KUKA KRL data list: tcp_chk_1.dat

&ACCESS RVP
&REL 151
&COMMENT TCP CHECK TOOL 1
DEFDAT  TCP_CHK_1
;FOLD EXTERNAL DECLARATIONS;%{PE}%V3.2.0,%MKUKATPBASIS,%CEXT,%VCOMMON,%P
;FOLD GRIPPERTECH EXT
EXT  H50 (INT  :IN,INT  :IN,INT  :IN,GRP_TYP  :IN )
;ENDFOLD (GRIPPERTECH EXT)
;FOLD SPOTTECH EXT
EXT  USERSPOT (S_COMMAND  :IN,SPOT_TYPE  :IN )
;ENDFOLD (SPOTTECH EXT)
;FOLD BAS EXT;%{PE}%V3.2.0,%MKUKATPBASIS,%CEXT,%VEXT,%P
EXT  BAS (BAS_COMMAND  :IN,REAL  :IN )
DECL INT SUCCESS
;ENDFOLD
;FOLD USER EXT;%{E}%V3.2.0,%MKUKATPUSER,%CEXT,%VEXT,%P
;Make here your modifications
;ENDFOLD
;ENDFOLD
;FOLD USER EXT;%{}%V2.2.2,%MKUKATPUSER,%CEXT,%VEXT,%P
;Make here your modifications
DECL BOOL TIPKONTROLE
DECL INT ANSWER
DECL INT WAITTIME=1000
;ENDFOLD
;ENDFOLD
DECL INT I
;*      FDAT Declarations     *

;******************************
;*     E6POS Declarations     *
;******************************

DECL E6POS XP10={X 1991.58301,Y -779.688782,Z 1569.90405,A -142.057907,B 56.2479897,C -135.499695,S 2,T 2,E1 0.0,E2 0.0,E3 0.0,E4 0.0,E5 0.0,E6 0.0}
DECL E6POS XSERV_POS_1={X 84.4434509,Y 1847.146,Z 1622.83398,A 86.5612411,B -12.4712801,C -179.259094,S 6,T 27,E1 -1563.58301,E2 0.0,E3 0.0,E4 0.0,E5 0.0,E6 0.0}
DECL E6POS XP20={X 1368.17004,Y -1604.78003,Z 695.290527,A -176.796097,B 21.8214397,C -158.206604,S 2,T 2,E1 0.0,E2 0.0,E3 0.0,E4 0.0,E5 0.0,E6 0.0}

;******************************
;*     FDAT Declarations      *
;******************************

DECL FDAT FP10={TOOL_NO 14,BASE_NO 0,IPO_FRAME #BASE,TQ_STATE FALSE}
DECL FDAT FSERV_POS_1={TOOL_NO 1,BASE_NO 0,IPO_FRAME #BASE}
DECL FDAT FP20={TOOL_NO 14,BASE_NO 0,IPO_FRAME #BASE,TQ_STATE FALSE}

;******************************
;*  PDAT & LDAT Declarations  *
;******************************

DECL PDAT PH={VEL 100.0,ACC 100.0,APO_DIST 100.0,APO_MODE #CPTP}

DECL E6POS XP30={X 2311.08911,Y -615.218384,Z 582.254517,A 52.0533791,B 11.4944496,C -0.662933111,S 2,T 10,E1 -367.19989,E2 0.0,E3 0.0,E4 0.0,E5 0.0,E6 0.0}
DECL FDAT FP30={TOOL_NO 1,BASE_NO 0,IPO_FRAME #BASE,POINT2[] " "}
DECL E6POS XP40={X 2415.06006,Y -661.647217,Z -64.6423798,A 52.025631,B 13.8356104,C -0.669203103,S 2,T 8,E1 -367.19989,E2 0.0,E3 0.0,E4 0.0,E5 0.0,E6 0.0}
DECL FDAT FP40={TOOL_NO 1,BASE_NO 0,IPO_FRAME #BASE,POINT2[] " "}
DECL E6POS XP50={X 1079.88,Y -976.492493,Z 903.200806,A -177.984299,B 18.5442696,C -161.646393,S 2,T 2,E1 0.0,E2 0.0,E3 0.0,E4 0.0,E5 0.0,E6 0.0}
DECL FDAT FP50={TOOL_NO 0,BASE_NO 0,IPO_FRAME #BASE,POINT2[] " ",TQ_STATE FALSE}
DECL E6POS XP60={X 1368.17004,Y -1604.78003,Z 695.290527,A -176.796097,B 21.8214397,C -158.206604,S 2,T 2,E1 0.0,E2 0.0,E3 0.0,E4 0.0,E5 0.0,E6 0.0}
DECL FDAT FP60={TOOL_NO 14,BASE_NO 0,IPO_FRAME #BASE,POINT2[] " ",TQ_STATE FALSE}
DECL E6POS XP70={X 1991.58301,Y -779.688782,Z 1569.90405,A -142.057907,B 56.2479897,C -135.499695,S 2,T 2,E1 0.0,E2 0.0,E3 0.0,E4 0.0,E5 0.0,E6 0.0}
DECL FDAT FP70={TOOL_NO 14,BASE_NO 0,IPO_FRAME #BASE,POINT2[] " ",TQ_STATE FALSE}
DECL E6POS XP80={X 2192.04395,Y -596.577576,Z 555.076416,A -14.5445995,B 80.1722412,C -56.6474991,S 2,T 10,E1 -367.19989,E2 0.0,E3 0.0,E4 0.0,E5 0.0,E6 0.0}
DECL FDAT FP80={TOOL_NO 1,BASE_NO 0,IPO_FRAME #BASE,POINT2[] " "}
DECL E6POS XTCP_CHK_POSITION={X 84.4434509,Y 1847.146,Z 1622.83398,A 86.5612411,B -12.4712801,C -179.259094,S 6,T 27,E1 -1563.58301,E2 0.0,E3 0.0,E4 0.0,E5 0.0,E6 0.0}
DECL FDAT FTCP_CHK_POSITION={TOOL_NO 1,BASE_NO 0,IPO_FRAME #BASE,POINT2[] " "}
DECL E6POS XTCP_CHK_POS_1={X 818.403015,Y -1651.55701,Z -109.656601,A 172.554398,B -1.01382303,C -179.870605,S 2,T 2,E1 0.0,E2 0.0,E3 0.0,E4 0.0,E5 0.0,E6 0.0}
DECL FDAT FTCP_CHK_POS_1={TOOL_NO 14,BASE_NO 0,IPO_FRAME #BASE,POINT2[] " ",TQ_STATE FALSE}
DECL E6POS XP41={X 2432.96289,Y -476.577606,Z -71.2344208,A 52.0531807,B 11.4962101,C -0.664697111,S 2,T 8,E1 -367.19989,E2 0.0,E3 0.0,E4 0.0,E5 0.0,E6 0.0}
DECL FDAT FP41={TOOL_NO 1,BASE_NO 0,IPO_FRAME #BASE,POINT2[] " "}
DECL E6POS XP81={X 1822.90698,Y -654.884888,Z 640.681885,A 41.8054695,B 56.6090698,C 47.6876106,S 6,T 26,E1 -1972.61694,E2 0.0,E3 0.0,E4 0.0,E5 0.0,E6 0.0}
DECL FDAT FP81={TOOL_NO 1,BASE_NO 0,IPO_FRAME #BASE,POINT2[] " "}
DECL E6POS XBefore_Check_Point_1={X 818.62738,Y -1651.66101,Z -32.1126099,A 172.352905,B -1.31993604,C -179.733002,S 2,T 2,E1 0.0,E2 0.0,E3 0.0,E4 0.0,E5 0.0,E6 0.0}
DECL FDAT FBefore_Check_Point_1={TOOL_NO 14,BASE_NO 0,IPO_FRAME #BASE,POINT2[] " ",TQ_STATE FALSE}
DECL LDAT LH={VEL 2.0,ACC 100.0,APO_DIST 100.0,APO_FAC 50.0,ORI_TYP #VAR}
DECL E6POS XAFTER_CHECK_POINT_1={X 818.401428,Y -1651.55701,Z 10.4140701,A 172.554199,B -1.01384497,C -179.870697,S 2,T 2,E1 0.0,E2 0.0,E3 0.0,E4 0.0,E5 0.0,E6 0.0}
DECL FDAT FAfter_Check_Point_1={TOOL_NO 14,BASE_NO 0,IPO_FRAME #BASE,POINT2[] " ",TQ_STATE FALSE}
DECL E6POS XP75={X 2305.34692,Y -723.78302,Z 579.621582,A -14.5605898,B 80.1713333,C -56.66325,S 2,T 10,E1 -367.19989,E2 0.0,E3 0.0,E4 0.0,E5 0.0,E6 0.0}
DECL FDAT FP75={TOOL_NO 1,BASE_NO 0,IPO_FRAME #BASE,POINT2[] " "}
DECL E6POS XP90={X 2410.20093,Y -416.701294,Z 388.115906,A -122.975998,B 80.2214584,C -160.4422,S 2,T 10,E1 -422.983612,E2 0.0,E3 0.0,E4 0.0,E5 0.0,E6 0.0}
DECL FDAT FP90={TOOL_NO 1,BASE_NO 0,IPO_FRAME #BASE,POINT2[] " "}
DECL E6POS XBefore_Check_Point_2={X 2377.53491,Y -467.046295,Z 39.8671989,A -122.976303,B 80.2215729,C -160.442596,S 2,T 10,E1 -422.983612,E2 0.0,E3 0.0,E4 0.0,E5 0.0,E6 0.0}
DECL FDAT FBefore_Check_Point_2={TOOL_NO 1,BASE_NO 0,IPO_FRAME #BASE,POINT2[] " "}
DECL E6POS XTCP_CHK_POS_2={X 2426.96411,Y -429.442688,Z 29.7570896,A -126.074799,B 78.3430786,C -164.518799,S 2,T 10,E1 -422.981812,E2 0.0,E3 0.0,E4 0.0,E5 0.0,E6 0.0}
DECL FDAT FTCP_CHK_POS_2={TOOL_NO 1,BASE_NO 0,IPO_FRAME #BASE,POINT2[] " "}
DECL E6POS XAfter_Check_Point_2={X 2377.53491,Y -467.046295,Z 39.8671989,A -122.976303,B 80.2215729,C -160.442596,S 2,T 10,E1 -422.983612,E2 0.0,E3 0.0,E4 0.0,E5 0.0,E6 0.0}
DECL FDAT FAfter_Check_Point_2={TOOL_NO 1,BASE_NO 0,IPO_FRAME #BASE,POINT2[] " "}
DECL E6POS XP100={X 2410.19995,Y -416.696594,Z 388.11441,A -122.976501,B 80.2214966,C -160.442795,S 2,T 10,E1 -422.985291,E2 0.0,E3 0.0,E4 0.0,E5 0.0,E6 0.0}
DECL FDAT FP100={TOOL_NO 1,BASE_NO 0,IPO_FRAME #BASE,POINT2[] " "}
DECL E6POS XP110={X 1784.026,Y -939.821716,Z 564.808594,A -112.103302,B 88.3751907,C -136.251404,S 2,T 10,E1 -586.802917,E2 0.0,E3 0.0,E4 0.0,E5 0.0,E6 0.0}
DECL FDAT FP110={TOOL_NO 1,BASE_NO 0,IPO_FRAME #BASE,POINT2[] " "}
DECL E6POS XP120={X 996.789307,Y -1256.22302,Z 985.020386,A -19.8349094,B 83.8573227,C -28.9672508,S 2,T 10,E1 -831.47522,E2 0.0,E3 0.0,E4 0.0,E5 0.0,E6 0.0}
DECL FDAT FP120={TOOL_NO 1,BASE_NO 0,IPO_FRAME #BASE,POINT2[] " "}
DECL E6POS XP130={X 605.816284,Y -317.149902,Z 1161.85999,A 86.4495468,B 72.0065536,C 88.4566193,S 6,T 26,E1 -1309.93506,E2 0.0,E3 0.0,E4 0.0,E5 0.0,E6 0.0}
DECL FDAT FP130={TOOL_NO 1,BASE_NO 0,IPO_FRAME #BASE,POINT2[] " "}
DECL SPOT_SUGG_T LAST_SPOT={GUN[] "1                       ",RETR_CMD[] "#CLO                    ",CHOISE[] "#FIRST                  ",CLO_TM[] "0                       ",PGNO1[] "1                       ",PRESS1[] "0                       ",PGNO2[] "1                       ",PRESS2[] "0                       ",SPOT_PARAMS[] "SDAT0                   "}
DECL BASIS_SUGG_T LAST_BASIS={POINT1[] "P21                     ",POINT2[] "P21                     ",CP_PARAMS[] "CPDAT2                  ",PTP_PARAMS[] "PDAT8                   ",CONT[] "                        ",CP_VEL[] "0.5                     ",PTP_VEL[] "100                     ",SYNC_PARAMS[] "SYNCDAT                 ",SPL_NAME[] "S0                      "}
DECL E6POS XP140={X 561.656921,Y -133.506302,Z 985.631287,A 133.0784,B 72.5561295,C -179.839905,S 6,T 26,E1 -1972.61096,E2 0.0,E3 0.0,E4 0.0,E5 0.0,E6 0.0}
DECL FDAT FP140={TOOL_NO 1,BASE_NO 0,IPO_FRAME #BASE,POINT2[] " "}
DECL PDAT PPDAT2={VEL 100.0,ACC 100.0,APO_DIST 100.0,APO_MODE #CPTP}
DECL E6POS XP11={X -805.688477,Y 970.449097,Z 1769.79395,A 53.8147697,B -6.02124786,C -157.374298,S 2,T 3,E1 0.0,E2 0.0,E3 0.0,E4 0.0,E5 0.0,E6 0.0}
DECL FDAT FP11={TOOL_NO 0,BASE_NO 0,IPO_FRAME #BASE,POINT2[] " ",TQ_STATE FALSE}
DECL PDAT PPDAT3={VEL 100.0,ACC 100.0,APO_DIST 100.0,APO_MODE #CPTP}
DECL E6POS XP12={X -1121.82495,Y 605.006226,Z 1520.71802,A 95.0571289,B -0.001507523,C 179.989899,S 2,T 3,E1 0.0,E2 0.0,E3 0.0,E4 0.0,E5 0.0,E6 0.0}
DECL FDAT FP12={TOOL_NO 0,BASE_NO 0,IPO_FRAME #BASE,POINT2[] " ",TQ_STATE FALSE}
DECL LDAT LCPDAT0={VEL 2.0,ACC 100.0,APO_DIST 100.0,APO_FAC 50.0,ORI_TYP #VAR,CIRC_TYP #BASE,JERK_FAC 50.0,EXAX_IGN 0}
DECL E6POS XP13={X -1121.80103,Y 605.010803,Z 1376.47803,A 95.0571136,B -0.00151944801,C 179.990005,S 2,T 3,E1 0.0,E2 0.0,E3 0.0,E4 0.0,E5 0.0,E6 0.0}
DECL FDAT FP13={TOOL_NO 0,BASE_NO 0,IPO_FRAME #BASE,POINT2[] " ",TQ_STATE FALSE}
DECL LDAT LCPDAT1={VEL 2.0,ACC 100.0,APO_DIST 100.0,APO_FAC 50.0,ORI_TYP #VAR,CIRC_TYP #BASE,JERK_FAC 50.0,EXAX_IGN 0}
DECL E6POS XP14={X -1121.82495,Y 605.006226,Z 1520.71802,A 95.0571289,B -0.001507523,C 179.989899,S 2,T 3,E1 0.0,E2 0.0,E3 0.0,E4 0.0,E5 0.0,E6 0.0}
DECL FDAT FP14={TOOL_NO 0,BASE_NO 0,IPO_FRAME #BASE,POINT2[] " ",TQ_STATE FALSE}
DECL PDAT PPDAT4={VEL 100.0,ACC 100.0,APO_DIST 100.0,APO_MODE #CPTP}
DECL E6POS XP15={X -805.688477,Y 970.449097,Z 1769.79395,A 53.8147697,B -6.02124786,C -157.374298,S 2,T 3,E1 0.0,E2 0.0,E3 0.0,E4 0.0,E5 0.0,E6 0.0}
DECL FDAT FP15={TOOL_NO 0,BASE_NO 0,IPO_FRAME #BASE,POINT2[] " ",TQ_STATE FALSE}
DECL PDAT PPDAT5={VEL 100.0,ACC 100.0,APO_DIST 100.0,APO_MODE #CPTP}
DECL E6POS XP16={X 1402.91003,Y -456.992401,Z 1553.34204,A 169.668106,B 14.2850199,C -177.814804,S 2,T 2,E1 0.0,E2 0.0,E3 0.0,E4 0.0,E5 0.0,E6 0.0}
DECL FDAT FP16={TOOL_NO 0,BASE_NO 0,IPO_FRAME #BASE,POINT2[] " ",TQ_STATE FALSE}
DECL PDAT PPDAT6={VEL 100.0,ACC 100.0,APO_DIST 100.0,APO_MODE #CPTP}
DECL E6POS XP17={X 1079.88,Y -976.492493,Z 903.200806,A -177.984299,B 18.5442696,C -161.646393,S 2,T 2,E1 0.0,E2 0.0,E3 0.0,E4 0.0,E5 0.0,E6 0.0}
DECL FDAT FP17={TOOL_NO 0,BASE_NO 0,IPO_FRAME #BASE,POINT2[] " ",TQ_STATE FALSE}
DECL PDAT PPDAT7={VEL 100.0,ACC 100.0,APO_DIST 100.0}
DECL E6POS XP18={X -499.635406,Y 2147.92896,Z 1293.03198,A -75.6103516,B 0.00231015007,C 179.999496,S 2,T 11,E1 0.0,E2 0.0,E3 0.0,E4 0.0,E5 0.0,E6 0.0}
DECL FDAT FP18={TOOL_NO 0,BASE_NO 0,IPO_FRAME #BASE,POINT2[] " ",TQ_STATE FALSE}
DECL LDAT LCPDAT2={VEL 2.0,ACC 100.0,APO_DIST 100.0,APO_FAC 50.0,ORI_TYP #VAR,CIRC_TYP #BASE,JERK_FAC 50.0,EXAX_IGN 0}
DECL E6POS XP19={X -498.966705,Y 2148.29297,Z 1238.33203,A -75.5597534,B 0.00342605007,C 179.999603,S 2,T 11,E1 0.0,E2 0.0,E3 0.0,E4 0.0,E5 0.0,E6 0.0}
DECL FDAT FP19={TOOL_NO 0,BASE_NO 0,IPO_FRAME #BASE,POINT2[] " ",TQ_STATE FALSE}
DECL LDAT LCPDAT3={VEL 2.0,ACC 100.0,APO_DIST 100.0,APO_FAC 50.0,ORI_TYP #VAR,CIRC_TYP #BASE,JERK_FAC 50.0,EXAX_IGN 0}
DECL PDAT PPDAT8={VEL 100.0,ACC 100.0,APO_DIST 100.0,APO_MODE #CPTP}
DECL E6POS XP21={X 311.154999,Y 2009.28101,Z 1610.11304,A -96.3398895,B 10.9087496,C 179.568298,S 2,T 11,E1 0.0,E2 0.0,E3 0.0,E4 0.0,E5 0.0,E6 0.0}
DECL FDAT FP21={TOOL_NO 0,BASE_NO 0,IPO_FRAME #BASE,POINT2[] " ",TQ_STATE FALSE}
ENDDAT
